Yaskawa INFORM job: CALIBRATION_STANDARD.JBI

/JOB
//NAME CALIBRATION_STANDARD
//POS
///NPOS 20,0,0,0,0,0
///TOOL 0
///POSTYPE PULSE
///PULSE
C00000=208,-75312,1200,1,-127658,-69
C00001=-65160,-163660,-127880,-27700,-57282,17604
C00002=-113924,37261,-15839,-53976,-37776,36022
C00003=-88935,71842,22776,-38328,-30113,23127
C00004=118388,64274,14120,47959,-74513,-50857
C00005=75149,-145859,-123958,43122,-68431,-32519
C00006=42804,-31159,-73294,53963,-32933,-35202
C00007=148382,-75311,1200,0,-127658,-70
C00008=-154802,-75311,1200,0,-127658,-70
C00009=206,-2208,1200,0,-127658,-70
C00010=206,-166566,1200,0,-127658,-70
C00011=206,-75311,123177,0,-127658,-70
C00012=206,-75311,-86954,0,-127658,-70
C00013=206,-75311,1200,153424,-127658,-70
C00014=206,-75311,1200,-153424,-127658,-70
C00015=206,-75311,1196,0,5700,-72
C00016=206,-75312,1196,0,-132260,-71
C00017=206,-75311,1200,0,-127658,109912
C00018=206,-75311,1200,0,-127658,-109925
C00019=-77633,-75310,1200,0,-127658,-70
//INST
///DATE 2026/08/24 08:33
///ATTR SC,RW
///GROUP1 RB1
NOP
'1 HOME POSTION
MOVL C00000 V=423.3
'2 UF#2 S1 ORG
MOVL C00001 V=423.3
'3 UF#2 S1 RXX
MOVL C00002 V=423.3
'4 UF#2 S1 RXY
MOVL C00003 V=423.3
'5 UF#3 S2 ORG
MOVL C00004 V=423.3
'6 UF#3 S2 RXX
MOVL C00005 V=423.3
'7 UF#3 S2 RXY
MOVL C00006 V=423.3
'8 S+ SAFE LIMIT FROM HOME
MOVL C00007 V=423.3
'9 S- SAFE LIMIT FROM HOME
MOVL C00008 V=423.3
'10 L+ SAFE LIMIT FROM HOME
MOVL C00009 V=423.3
'11 L- SAFE LIMIT FROM HOME
MOVL C00010 V=423.3
'12 U+ SAFE LIMIT FROM HOME
MOVL C00011 V=423.3
'13 U- SAFE LIMIT FROM HOME
MOVL C00012 V=423.3
'14 R+ SAFE LIMIT FROM HOME
MOVL C00013 V=423.3
'15 R- SAFE LIMIT FROM HOME
MOVL C00014 V=423.3
'16 B+ SAFE LIMIT FROM HOME
MOVL C00015 V=423.3
'17 B- SAFE LIMIT FROM HOME
MOVL C00016 V=423.3
'18 T+ SAFE LIMIT FROM HOME
MOVL C00017 V=423.3
'19 T- SAFE LIMIT FROM HOME
MOVL C00018 V=423.3
'20 EXTRA CLEAR POSE
MOVL C00019 V=423.3
END
